{attribute 'qualified_only'}
VAR_GLOBAL
	station:typeStation; //data relating to the entire station
END_VAR

(* stored: Version 1.1.0.1, ProductVersion 3.1.4024.12
   GVL S2_Global: Id {f2ca5b31-1de6-4f3f-a24a-982c8035197d} *)
